// TIA Portal V17 export
// export: Created 2022-06-27T13:57:34.4170522Z, ExportSetting WithDefaults, DisplayName Totally Integrated Automation Portal, DisplayVersion V17 Update 3, DisplayName TIA Portal Openness, DisplayVersion V17 Update 3, DisplayName TIA Portal Version Control Interface, DisplayVersion V17, DisplayName SINAMICS Startdrive Advanced, DisplayVersion V17 Update1, DisplayName SINAMICS Startdrive G110M, G120, G120C, G120D, G120P, G115D, DisplayVersion V17 Update1, DisplayName SINAMICS Startdrive G130, G150, S120, S150, SINAMICS MV, S210, DisplayVersion V17 Update1, DisplayName STEP 7 Professional, DisplayVersion V17 Update 3, DisplayName STEP 7 Safety, DisplayVersion V17, DisplayName WinCC UA Professional, DisplayVersion V17 Update 3
FUNCTION_BLOCK "S04_MOTORS"   // FB4, LAD
{ S7_Optimized_Access := 'TRUE' }
VERSION : 0.1
// stored: AutoNumber false, IsIECCheckEnabled false, IsRetainMemResEnabled false, MemoryReserve 100, SetENOAutomatically false, UDAEnableTagReadback false
   VAR
      S041_DIRECT_START_MOTOR_Instance { S7_SetPoint := 'True'} : "S041_DIRECT_START_MOTOR";
      S042_DRIVER_MOTOR_Instance { S7_SetPoint := 'True'} : "S042_DRIVER_MOTOR";
      FB_MOTOR_SEQUENCE_STARTER_Instance { S7_SetPoint := 'True'} : "FB_MOTOR_SEQUENCE_STARTER";
   END_VAR
BEGIN

REGION Network 1: Call Motor sequence starter
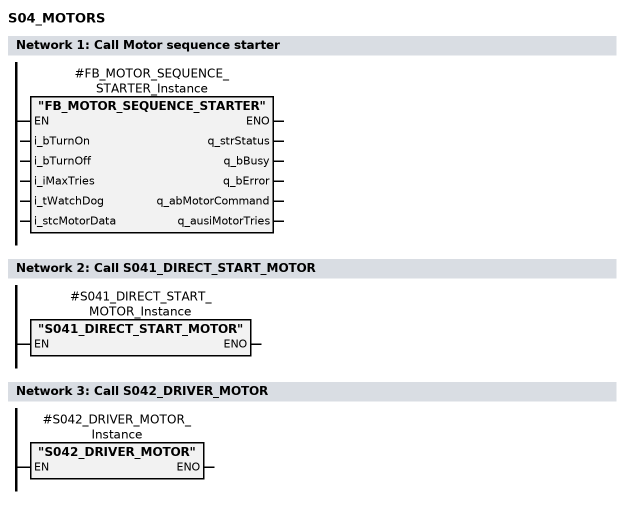
   RUNG wire#powerrail
      #FB_MOTOR_SEQUENCE_STARTER_Instance(i_bTurnOn :=, i_bTurnOff :=, i_iMaxTries :=, i_tWatchDog :=, i_stcMotorData :=, q_strStatus =>, q_bBusy =>, q_bError =>, q_abMotorCommand =>, q_ausiMotorTries =>)
   END_RUNG
   // the same network as SCL:
   #FB_MOTOR_SEQUENCE_STARTER_Instance();   // "FB_MOTOR_SEQUENCE_STARTER"
END_REGION

REGION Network 2: Call S041_DIRECT_START_MOTOR
   RUNG wire#powerrail
      #S041_DIRECT_START_MOTOR_Instance()
   END_RUNG
   // the same network as SCL:
   #S041_DIRECT_START_MOTOR_Instance();   // "S041_DIRECT_START_MOTOR"
END_REGION

REGION Network 3: Call S042_DRIVER_MOTOR
   RUNG wire#powerrail
      #S042_DRIVER_MOTOR_Instance()
   END_RUNG
   // the same network as SCL:
   #S042_DRIVER_MOTOR_Instance();   // "S042_DRIVER_MOTOR"
END_REGION
END_FUNCTION_BLOCK
